KUKA KRL data list: auto_mode.dat

&ACCESS RV
DEFDAT auto_mode PUBLIC

ENDDAT
